// TIA Portal V19 export
TYPE "LSNTP_typeTelegram"
// stored: Access Published
   STRUCT
      flags : Array[0..3] of Byte;   // Leap inidcator, version, mode, stratum, poll, precision
      rootDelay : DWord;   // Indicates the total round trip delay to the primary reference source in seconds
      rootDispersion : DWord;   // Indicates the maximum error due to the clock frequency tolerance
      referenceId : Array[0..3] of Char;   // Identifies the clock reference source
      timestamps : Struct   // Timestamps
         reference { S7_SetPoint := 'True'} : "LSNTP_typeTimestamp";   // Time when the system clock was last set or corrected
         originate { S7_SetPoint := 'True'} : "LSNTP_typeTimestamp";   // Time when the request departed the client
         receive { S7_SetPoint := 'True'} : "LSNTP_typeTimestamp";   // Time when the server received the request
         transmit { S7_SetPoint := 'True'} : "LSNTP_typeTimestamp";   // Time when the reply departed the server
      END_STRUCT;
      keyIdentifier : DWord;   // (Optional) Contains the message authentication code if authentication scheme is implemented
      messageDigest : Array[0..15] of Byte;   // (Optional) Contains the message authentication code if authentication scheme is implemented
   END_STRUCT;
END_TYPE
